{attribute 'enable_dynamic_creation'}
FUNCTION_BLOCK FB_A
VAR
	value : BOOL;
	value2 : REAL := 42;
END_VAR

METHOD Sum : INT
VAR_INPUT
	value1 : INT;
	value2: INT;
END_VAR
Sum := value1 + value2;
END_METHOD

END_FUNCTION_BLOCK

(* stored: Version 1.1.0.1, ProductVersion 3.1.4024.12
   POU FB_A: Id {44e90c3b-96dc-4e5b-9818-b1ed8f01a501}, SpecialFunc None
   Method Sum: Id {fdb674d3-65b4-453a-a482-05eccfc2ab42} *)
